// The verdict cannot return to Passed once a check has failed. Later checks are

// still evaluated and counted - a run should report everything it found, not stop

// at the first problem - but none of them can undo the first failure.
FUNCTION_BLOCK TEST_VerdictPassDoesNotOvertakeAFailure IMPLEMENTS I_Test
VAR
	// A private journal and handle, so a DELIBERATE failure can be recorded and

	// inspected without the suite's own verdict ever seeing it. The test itself

	// passes; what it proves is that failing works.
	Subject		   : TestJournal;
	Handle		   : TestVerdict;
	Same		   : DINT := 7;
	Lower		   : DINT := 1;
	Higher		   : DINT := 2;
	ExpectedStatus : E_TestStatus;
	ActualStatus   : E_TestStatus;
	ExpectedCount  : UDINT;
	ActualCount	   : UDINT;
END_VAR

METHOD Run : BOOL
VAR_INPUT
	Enable : BOOL;
	Test   : I_TestAssertions;
END_VAR
Handle.Target(Subject);
Subject.Begin('deliberate', '');
Handle.AssertEqual(Lower, Higher, 'fails first');
Handle.AssertEqual(Same, Same, 'passes second');
Handle.AssertTrue(TRUE, 'passes third');
ExpectedCount := 3;
ActualCount	  := Subject.AssertionCount;
Test.AssertEqual(ExpectedCount, ActualCount, 'every check was evaluated');
Subject.Finish(E_TestStatus.Passed);
ExpectedStatus := E_TestStatus.Failed;
ActualStatus   := Subject.Status;
Test.AssertEqual(ExpectedStatus, ActualStatus, 'still Failed after two passes');
Handle.Untarget();
Run := TRUE;
END_METHOD

END_FUNCTION_BLOCK

(* stored: Version 1.1.0.1, ProductVersion 3.1.4026.18
   POU TEST_VerdictPassDoesNotOvertakeAFailure: Id {c095c34a-45bf-4a15-ba30-e6cd3e183723}, SpecialFunc None
   Folder I_Test: Id {c346e70c-99c9-47e9-b60e-dd6f68444785}
   Method Run: Id {9122bd42-d0a6-4713-8e7b-6ba4aa149d9c} *)
